{region '#Template'}
	{attribute 'Category' := 'AC'}
	{attribute 'Version' := '0.0.1.0'}
	{attribute 'Tags' := 'AC, Aggregates, Pre-heater, Temperature, Controller'}
	{attribute 'Description' := 'Vorerhitzer Zuluft Regler Temperatur	// Pre-heater Supply air controller temperature'}
{endregion}
FUNCTION_BLOCK FB_BA_AC_PreHtrTSuACtrl EXTENDS FB_BA_View
VAR_INPUT
	bEn						: BOOL;
	fSpTSuA					: REAL;
	fTSuA					: REAL;
	bSync					: BOOL;
	fSync					: REAL;
	bDeHum					: BOOL;
END_VAR
VAR_OUTPUT
	fY              		: REAL;
	bIsActive				: BOOL;	//	active sequence controller
	bOpState				: BOOL;	//	Release sequence link, sequence control is active	
END_VAR
VAR_INPUT CONSTANT
	Ctrl					: FB_BA_Loop;	
END_VAR
VAR
	srDeHum					: SR;
	ftrigDeHum				: F_TRIG;
	rtrigSync				: R_TRIG;
	PrioSwiSync				: FB_BA_PrioSwi_R04;
END_VAR
VAR // added by the converter: edge detectors and wires of the graphical bodies
    _w1 : BOOL;
END_VAR

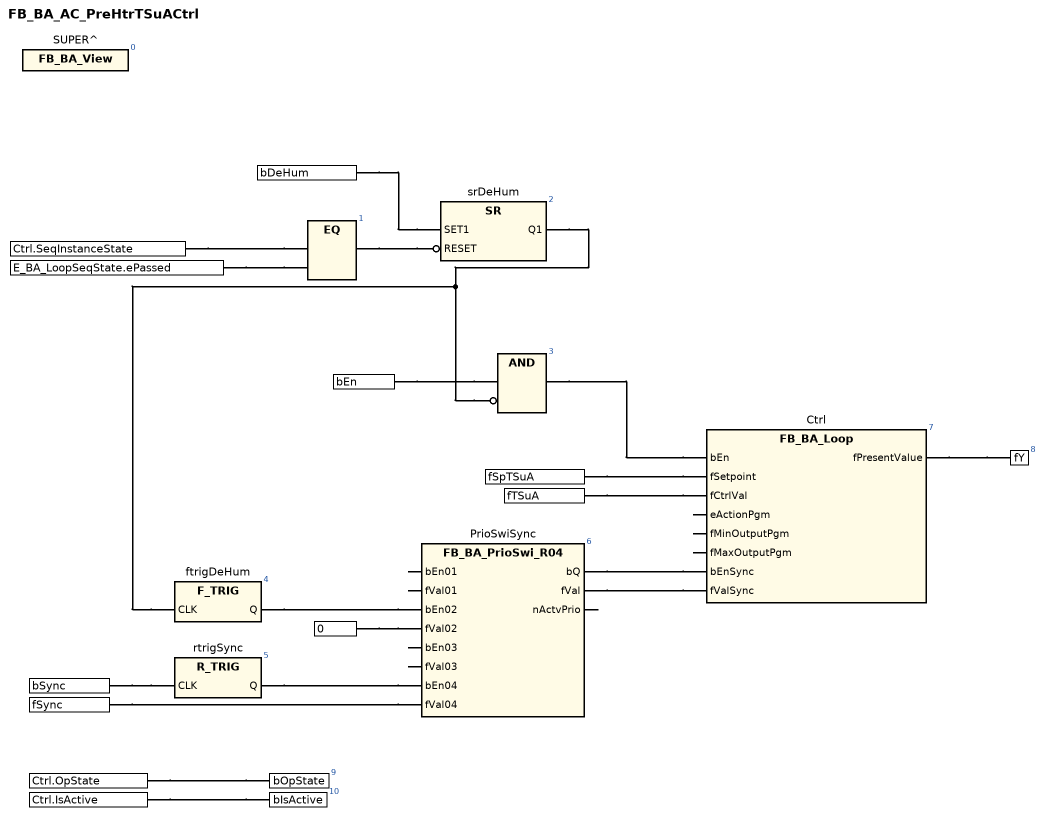
SUPER^(); // FB_BA_View
srDeHum(SET1 := bDeHum, RESET := NOT (Ctrl.SeqInstanceState = E_BA_LoopSeqState.ePassed)); // SR
_w1 := bEn AND NOT srDeHum.Q1;
ftrigDeHum(CLK := srDeHum.Q1); // F_TRIG
rtrigSync(CLK := bSync); // R_TRIG
PrioSwiSync(bEn02 := ftrigDeHum.Q, fVal02 := 0, bEn04 := rtrigSync.Q, fVal04 := fSync); // FB_BA_PrioSwi_R04
// parameter Ctrl.fIntegralConstant := 60
// parameter Ctrl.fProportionalConstant := 5
// parameter Ctrl.eActionRm := E_BA_Action.eReverse
Ctrl(
    bEn := _w1,
    fSetpoint := fSpTSuA,
    fCtrlVal := fTSuA,
    bEnSync := PrioSwiSync.bQ,
    fValSync := PrioSwiSync.fVal); // FB_BA_Loop
fY := Ctrl.fPresentValue;
bOpState := Ctrl.OpState;
bIsActive := Ctrl.IsActive;

METHOD FB_init : BOOL
VAR_INPUT
	bInitRetains : BOOL; // if TRUE, the retain variables are initialized (warm start / cold start)
	bInCopyCode : BOOL;  // if TRUE, the instance afterwards gets moved into the copy code (online change)
END_VAR
Ctrl.iParent						:= THIS^;
Ctrl.iLabel							:= LblCmpAC.PreHtr_TSuACtrl_Ctrl; 
Ctrl.sObjectName					:= '{Idx=01}';
Ctrl.eOpMode						:= BA2_Param.nLoop_DefOpMode;								 	 										 
Ctrl.eOutputUnit					:= E_BA_Unit.eOther_Percent;
Ctrl.eActionRm						:= E_BA_Action.eReverse;
Ctrl.fProportionalConstant			:= 3;
Ctrl.fIntegralConstant				:= 180;
Ctrl.fDerivativeConstant			:= 0;
Ctrl.fMaxOutputRm 					:= 100;
Ctrl.fMinOutputRm					:= 0;
Ctrl.fCOVIncrement					:= 0;
Ctrl.nDampConstant					:= 0;
Ctrl.fNeutralZone					:= 0;
Ctrl.stStepDelay.nDown				:= 0;
Ctrl.stStepDelay.nUp				:= 0;
END_METHOD

END_FUNCTION_BLOCK

(* stored: Version 1.1.0.1, ProductVersion 3.1.4024.6
   POU FB_BA_AC_PreHtrTSuACtrl: Id {dd6ac758-c2b9-4eb3-9821-ed5990c83680}, SpecialFunc None
   Method FB_init: Id {b1f60c2a-5952-4fac-97f5-55b4d8b50af5} *)
